FUNCTION_BLOCK PendingResponseMiddleware EXTENDS MiddlewareBase
VAR
	pendingResponseManager : I_PendingResponseManager;
END_VAR

METHOD FB_init : BOOL
VAR_INPUT
	bInitRetains : BOOL; // if TRUE, the retain variables are initialized (warm start / cold start)
	bInCopyCode : BOOL;  // if TRUE, the instance afterwards gets moved into the copy code (online change)
	PendingResponseManager : I_PendingResponseManager;
END_VAR
This^.pendingResponseManager := PendingResponseManager;
END_METHOD

METHOD PUBLIC Handle
VAR_INPUT
	Request : I_Request;
	Response : I_ServerResponse;
END_VAR
IF pendingResponseManager.TryHandleIncomingRequest(Request, Response) THEN
	RETURN;
END_IF

Next(Request, Response);
END_METHOD

END_FUNCTION_BLOCK

(* stored: Version 1.1.0.1, ProductVersion 3.1.4024.12
   POU PendingResponseMiddleware: Id {6371efe8-c6db-4885-801d-1a3c9cf89e08}, SpecialFunc None
   Folder Constructor: Id {86f52e50-6c9b-4a40-9d00-4b7da94a288c}
   Method FB_init: Id {a579fcf9-c9e3-4999-b21a-9e34ea053d3c}
   Method Handle: Id {8696b458-a0eb-4d91-a059-aff474e59f3b} *)
